(* PLC project Unnamed, Unknown Unnamed 1 *)
(* stored: creationDateTime 2017-02-14T17:58:59, modificationDateTime 2017-03-06T21:20:49 *)

TYPE CalType : REAL := 5.0;
END_TYPE

FUNCTION Norm : REAL
  VAR_INPUT
    BIK : SINT;
    LCtrlK : SINT;
    MType : BOOL;
  END_VAR
  VAR
    Calib : CalType;
    Type1 : REAL := 6.0;
    Type2 : REAL := 4.0;
  END_VAR

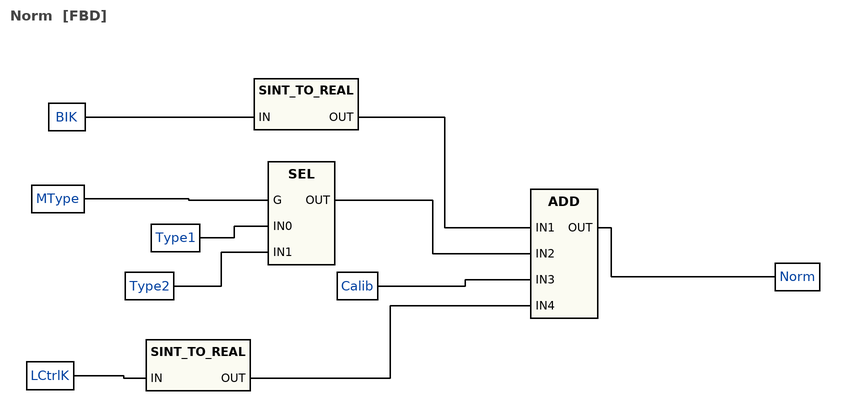
(* FBD diagram, written out as Structured Text *)
Norm := SINT_TO_REAL(BIK) + SEL(MType, Type1, Type2) + Calib + SINT_TO_REAL(LCtrlK);
END_FUNCTION

FUNCTION_BLOCK Volume
  VAR_INPUT
    BalControl : SINT;
    BalFactor : SINT := 5;  (* fasfasfaf *)
    VolControl : SINT;  (* ado *)
    ModelType : BOOL;
  END_VAR
  VAR_OUTPUT
    RightAmplif : REAL;
    LeftAmplif : REAL;
    LED : BOOL;
  END_VAR
  VAR_IN_OUT
    Critical : BOOL;
  END_VAR
  VAR CONSTANT
    MaxVolume : REAL := 26.0;
  END_VAR
  VAR
    Timeout : TIME := 2;
    HeatTime : TON;
    Overdrive : BOOL;
  END_VAR
  VAR  (* added by the conversion: wires and edge detectors of the diagram *)
    _Norm2_OUT : REAL;
    _Norm3_OUT : REAL;
  END_VAR

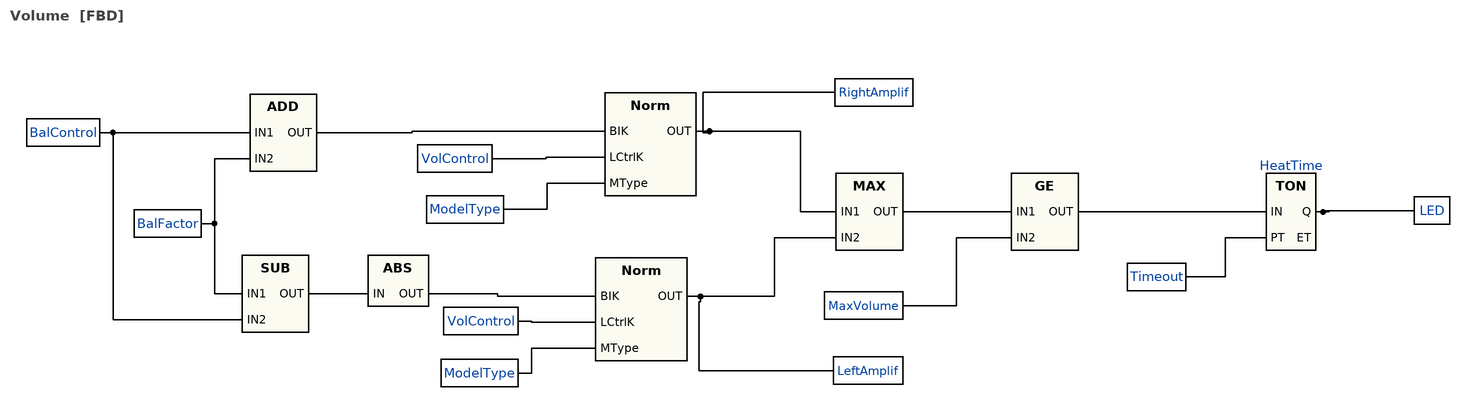
(* FBD diagram, written out as Structured Text *)
_Norm2_OUT := Norm(BalControl + BalFactor, VolControl, ModelType);
RightAmplif := _Norm2_OUT;
_Norm3_OUT := Norm(ABS(BalFactor - BalControl), VolControl, ModelType);
HeatTime(IN := MAX(_Norm2_OUT, _Norm3_OUT) >= MaxVolume, PT := Timeout);
LED := HeatTime.Q;
LeftAmplif := _Norm3_OUT;
END_FUNCTION_BLOCK

CONFIGURATION config
  RESOURCE resource0 ON PLC
  END_RESOURCE
END_CONFIGURATION
